(* IEC 61131-3 sources: com.logicals.lc3.webinar/usRTS_RPMControl_iSOC/src_FB_LIB_SAFE/Numeric/SINT, 8 files *)

(* ---- wADD_SINT_2.iecst ---- *)
NAMESPACE logicals.web.standard
NAMESPACE numeric

/*
 * Function block wrapper for IEC 61131-3 ADD<br>
 * IN1 =  1st value (SINT)<br>
 * IN2 =  2nd value (SINT)<br>
 * OUT = Sum of all input values (SINT)<br>
 */
FUNCTION_BLOCK wADD_SINT_2
	{ vNameAlignment:="center"; altName:="+"; bgColor:="LightPink"; width:=40; hideIONames; }
	VAR_INPUT
		IN1 : SINT;
		IN2 : SINT;
	END_VAR
	VAR_OUTPUT
		OUT : SINT;
	END_VAR

	OUT := ADD(IN1:=IN1, IN2:=IN2, ENO=>ENO);
END_FUNCTION_BLOCK

END_NAMESPACE
END_NAMESPACE

(* ---- wADD_SINT_3.iecst ---- *)
NAMESPACE logicals.web.standard
NAMESPACE numeric

/*
 * Function block wrapper for IEC 61131-3 ADD<br>
 * IN1 =  1st value (SINT)<br>
 * IN2 =  2nd value (SINT)<br>
 * IN3 =  3rd value (SINT)<br>
 * OUT = Sum of all input values (SINT)<br>
 */
FUNCTION_BLOCK wADD_SINT_3
	{ vNameAlignment:="center"; altName:="+"; bgColor:="LightPink"; width:=40; hideIONames; }
	VAR_INPUT
		IN1 : SINT;
		IN2 : SINT;
		IN3 : SINT;
	END_VAR
	VAR_OUTPUT
		OUT : SINT;
	END_VAR

	OUT := ADD(IN1:=IN1, IN2:=IN2, IN3:=IN3, ENO=>ENO);
END_FUNCTION_BLOCK

END_NAMESPACE
END_NAMESPACE

(* ---- wADD_SINT_4.iecst ---- *)
NAMESPACE logicals.web.standard
NAMESPACE numeric

/*
 * Function block wrapper for IEC 61131-3 ADD<br>
 * IN1 =  1st value (SINT)<br>
 * IN2 =  2nd value (SINT)<br>
 * IN3 =  3rd value (SINT)<br>
 * IN4 =  4th value (SINT)<br>
 * OUT = Sum of all input values (SINT)<br>
 */
FUNCTION_BLOCK wADD_SINT_4
	{ vNameAlignment:="center"; altName:="+"; bgColor:="LightPink"; width:=40; hideIONames; }
	VAR_INPUT
		IN1 : SINT;
		IN2 : SINT;
		IN3 : SINT;
		IN4 : SINT;
	END_VAR
	VAR_OUTPUT
		OUT : SINT;
	END_VAR

	OUT := ADD(IN1:=IN1, IN2:=IN2, IN3:=IN3, IN4:=IN4, ENO=>ENO);
END_FUNCTION_BLOCK

END_NAMESPACE
END_NAMESPACE

(* ---- wDIV_SINT.iecst ---- *)
NAMESPACE logicals.web.standard
NAMESPACE numeric

/*
 * Function block wrapper for IEC 61131-3 DIV<br>
 * IN1 =  1st value (SINT)<br>
 * IN2 =  2nd value (SINT)<br>
 * OUT = quotient of IN1 divided by IN2 (SINT)<br>
 */
FUNCTION_BLOCK wDIV_SINT
	{ vNameAlignment:="center"; altName:="/"; bgColor:="LightPink"; width:=40; hideIONames; }
	VAR_INPUT
		IN1 : SINT;
		IN2 : SINT;
	END_VAR
	VAR_OUTPUT
		OUT : SINT;
	END_VAR

	OUT := DIV(IN1:=IN1, IN2:=IN2, ENO=>ENO);
END_FUNCTION_BLOCK

END_NAMESPACE
END_NAMESPACE

(* ---- wMUL_SINT_2.iecst ---- *)
NAMESPACE logicals.web.standard
NAMESPACE numeric

/*
 * Function block wrapper for IEC 61131-3 MUL<br>
 * IN1 =  1st value (SINT)<br>
 * IN2 =  2nd value (SINT)<br>
 * OUT = Product of multiplication of all inputs (SINT)<br>
 */
FUNCTION_BLOCK wMUL_SINT_2
	{ vNameAlignment:="center"; altName:="*"; bgColor:="LightPink"; width:=40; hideIONames; }
	VAR_INPUT
		IN1 : SINT;
		IN2 : SINT;
	END_VAR
	VAR_OUTPUT
		OUT : SINT;
	END_VAR

	OUT := MUL(IN1:=IN1, IN2:=IN2, ENO=>ENO);
END_FUNCTION_BLOCK

END_NAMESPACE
END_NAMESPACE

(* ---- wMUL_SINT_3.iecst ---- *)
NAMESPACE logicals.web.standard
NAMESPACE numeric

/*
 * Function block wrapper for IEC 61131-3 MUL<br>
 * IN1 =  1st value (SINT)<br>
 * IN2 =  2nd value (SINT)<br>
 * IN3 =  3rd value (SINT)<br>
 * OUT = Product of multiplication of all inputs (SINT)<br>
 */
FUNCTION_BLOCK wMUL_SINT_3
	{ vNameAlignment:="center"; altName:="*"; bgColor:="LightPink"; width:=40; hideIONames; }
	VAR_INPUT
		IN1 : SINT;
		IN2 : SINT;
		IN3 : SINT;
	END_VAR
	VAR_OUTPUT
		OUT : SINT;
	END_VAR

	OUT := MUL(IN1:=IN1, IN2:=IN2, IN3:=IN3, ENO=>ENO);
END_FUNCTION_BLOCK

END_NAMESPACE
END_NAMESPACE

(* ---- wMUL_SINT_4.iecst ---- *)
NAMESPACE logicals.web.standard
NAMESPACE numeric

/*
 * Function block wrapper for IEC 61131-3 MUL<br>
 * IN1 =  1st value (SINT)<br>
 * IN2 =  2nd value (SINT)<br>
 * IN3 =  3rd value (SINT)<br>
 * IN4 =  4th value (SINT)<br>
 * OUT = Product of multiplication of all inputs (SINT)<br>
 */
FUNCTION_BLOCK wMUL_SINT_4
	{ vNameAlignment:="center"; altName:="*"; bgColor:="LightPink"; width:=40; hideIONames; }
	VAR_INPUT
		IN1 : SINT;
		IN2 : SINT;
		IN3 : SINT;
		IN4 : SINT;
	END_VAR
	VAR_OUTPUT
		OUT : SINT;
	END_VAR

	OUT := MUL(IN1:=IN1, IN2:=IN2, IN3:=IN3, IN4:=IN4, ENO=>ENO);
END_FUNCTION_BLOCK

END_NAMESPACE
END_NAMESPACE

(* ---- wSUB_SINT.iecst ---- *)
NAMESPACE logicals.web.standard
NAMESPACE numeric

/*
 * Function block wrapper for IEC 61131-3 SUB<br>
 * IN1 =  1st value (SINT)<br>
 * IN2 =  2nd value (SINT)<br>
 * OUT = IN1 minus IN2 (SINT)<br>
 */
FUNCTION_BLOCK wSUB_SINT
	{ vNameAlignment:="center"; altName:="-"; bgColor:="LightPink"; width:=40; hideIONames; }
	VAR_INPUT
		IN1 : SINT;
		IN2 : SINT;
	END_VAR
	VAR_OUTPUT
		OUT : SINT;
	END_VAR

	OUT := SUB(IN1:=IN1, IN2:=IN2, ENO=>ENO);
END_FUNCTION_BLOCK

END_NAMESPACE
END_NAMESPACE
